{attribute 'qualified_only'}
VAR_GLOBAL
	//motion rows and buttons to feedback into program
	gMotionRows: typeMotionScreen;
	gMotionRowButtons: typeMotionScreenBtn;
END_VAR

(* stored: Version 1.1.0.1, ProductVersion 3.1.4024.12
   GVL gHMIMotionRows: Id {d58e2224-54a1-4417-8c42-c635c8255aee} *)
